// LS Electric XG5000 project: 2024.11.11.Fin_Project
// PLC LSPLC

PROGRAM NewProgram (task: 스캔 프로그램)

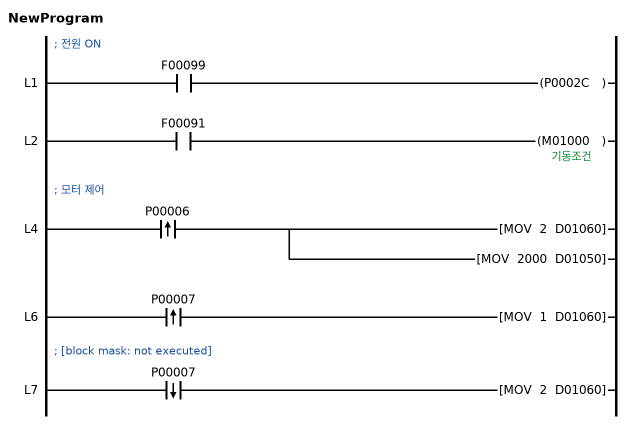
// 전원 ON
; L1
LOAD      F00099
OUT       P0002C
; L2
LOAD      F00091
OUT       M01000	// 기동조건
// 모터 제어
; L4
LOADP     P00006
MOV       2 D01060
MOV       2000 D01050
; L6
LOADP     P00007
MOV       1 D01060
; L7 (block mask: not executed)
LOADN     P00007
MOV       2 D01060